# B&R Automation Studio project lektion_6_agdp
Automation Studio 4.8.2.72

## Configuration Config1

### Hardware
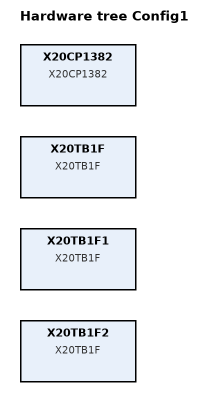
```
X20CP1382 : X20CP1382 v1.10.0.0  [X1 -> X1.SL; X2 -> X2.SL; X3 -> X3.SL]
  Module X1 (Type=X1, Virtual=true, Version=1.10.0.0)
    Connection (Connector=SS1, TargetModule=X20TB1F, TargetConnector=SS)
    Connection (Connector=SL, TargetModule=X20CP1382, TargetConnector=X1)
  Module X2 (Type=X2, Virtual=true, Version=1.10.0.0)
    Connection (Connector=SS1, TargetModule=X20TB1F1, TargetConnector=SS)
    Connection (Connector=SL, TargetModule=X20CP1382, TargetConnector=X2)
  Module X3 (Type=X3, Virtual=true, Version=1.10.0.0)
    Connection (Connector=SS1, TargetModule=X20TB1F2, TargetConnector=SS)
    Connection (Connector=SL, TargetModule=X20CP1382, TargetConnector=X3)
  Connector IF2:
    ActivateDevice = 1
  ConfigurationID = lektion_VI_agdp_Config1
  Simulation = 1
X20TB1F : X20TB1F v1.0.0.0
X20TB1F1 : X20TB1F v1.0.0.0
X20TB1F2 : X20TB1F v1.0.0.0
```

## Logical view

### Program Logical/Opg1

#### Main.st
```iecst
PROGRAM _INIT
	(* Insert code here *)

END_PROGRAM

PROGRAM _CYCLIC
	(* Insert code here *)
	A := A + 1;

END_PROGRAM

PROGRAM _EXIT
	(* Insert code here *)

END_PROGRAM
```

### Program Logical/Opg2

#### Variables.var
```iecst
VAR
	array : ARRAY[0..15] OF BOOL;
	shift : BOOL;
	i : USINT;
	tmp : BOOL;
END_VAR
```

#### Main.st
```iecst
PROGRAM _INIT
	(* Insert code here *)
	array[0] := TRUE;
	shift := TRUE;
END_PROGRAM

PROGRAM _CYCLIC
	(* Insert code here *)
	IF shift THEN
		tmp := array[0];
		array[0] := array[1];
		array[1] := array[2];
		array[2] := array[3];
		array[3] := array[4];
		array[4] := array[5];
		array[5] := array[6];
		array[6] := array[7];
		array[7] := array[8];
		array[8] := array[9];
		array[9] := array[10];
		array[10] := array[11];
		array[11] := array[12];
		array[12] := array[13];
		array[13] := array[14];
		array[14] := array[15];
		array[15] := tmp;
	END_IF;

END_PROGRAM

PROGRAM _EXIT
	(* Insert code here *)

END_PROGRAM
```
